TYPE UR_7_T2O_FloatRegisters :
STRUCT
	  Floats : ARRAY[0..23] OF REAL;
END_STRUCT
END_TYPE

(* stored: Version 1.1.0.1
   DUT UR_7_T2O_FloatRegisters: Id {6c1d8e2c-98fb-4573-aee9-defc0298f81c} *)
